// TwinCAT 3 PLC project MotionDriver
// ProgramVersion: 3.1.4026.20
// libraries:
//   Tc2_MC2, * (Beckhoff Automation GmbH)
//   Tc2_Standard, * (Beckhoff Automation GmbH)
//   Tc2_System, * (Beckhoff Automation GmbH)
// project tree:
//   GVLs/ gVar.TcGVL
//   / PlcTask.TcTTO
//   POUs/ AxisDriver.TcPOU
// real-time tasks:
//   TASK PlcTask: cycle T#1ms, priority 20, ADS port 350
// motion (NC):
//   TASK NC-Task 1 SAF: cycle T#500us, priority 1, ADS port 501
//   TASK NC-Task 1 SVB: cycle T#10ms, priority 8, ADS port 511
//   AXIS Axis 1 (id 1)
//     General: UnitName=Degree
//     Dynamic: AccelerationMaximum=500, DecelerationMaximum=500, Acceleration=300, Deceleration=300, Jerk=1300
//     Velo: Maximum=50
//     OtherSettings: AllowMotionCmdToSlave=true
//     encoder EncType=19
//       EncPara: MaxCount=#xffffffff
//     drive DrvType=16
//       DrvPara: MaxCount=#xffffffff, DriveControlDWord=#x00020000
//         Analog: VeloReferenz=50, TorqueSetpointScale=10, ScaleFactorActTorque=0.1
//         TimeComp: TaskDelayCycles=1
//     controller CtrType=1
//       CtrPara: PriorControlFactor=1
//         Observer: BandWidth=20
// I/O:
//   DEVICE IPC Master, AmsNetId 5.154.213.103.2.1
//     Drive 1 (CAP-NET-E) [CAP-NET-E]
// variable links:
//   NC-Task 1 SAF/Axes/Axis 1 <-> IPC Master/Drive 1 (CAP-NET-E)
//     Drive/Inputs/In/nState1 <-> TPDO 1 mapping parameter/Status Word
//     Drive/Inputs/In/nState2 <-> TPDO 1 mapping parameter/Status Word @bit 8
//     Drive/Inputs/In/nState4 @bit 1 <-> WcState/InputToggle
//     Drive/Inputs/In/nState4 <-> WcState/WcState
//     Drive/Inputs/In/nState5 <-> TPDO 1 mapping parameter/Modes of operation display
//     Drive/Outputs/Out/nCtrl1 <-> RPDO 1 mapping parameter/Control Word
//     Drive/Outputs/Out/nCtrl2 <-> RPDO 1 mapping parameter/Control Word @bit 8
//     Drive/Outputs/Out/nCtrl5 <-> RPDO 1 mapping parameter/Modes of operation
//     Drive/Outputs/Out/nDataOut1 <-> RPDO 1 mapping parameter/Target position
//     Drive/Outputs/Out/nDataOut2 <-> RPDO 1 mapping parameter/Target velocity
//     Enc/Inputs/In/nDataIn1 <-> TPDO 1 mapping parameter/Position actual value
//     Enc/Inputs/In/nDataIn7 <-> TPDO 1 mapping parameter/Velocity actual value
//     Enc/Inputs/In/nState4 @bit 1 <-> WcState/InputToggle
//     Enc/Inputs/In/nState4 <-> WcState/WcState
//   MotionDriver/MotionDriver Instance <-> NC-Task 1 SAF/Axes/Axis 1
//     PlcTask Inputs/gVar.gAxis1.NcToPlc <-> Outputs/ToPlc
//     PlcTask Outputs/gVar.gAxis1.PlcToNc <-> Inputs/FromPlc

CONFIGURATION MotionDriver
    RESOURCE PLC ON TwinCAT3
        TASK PlcTask(INTERVAL := T#1ms, PRIORITY := 20);
        PROGRAM AxisDriver WITH PlcTask : AxisDriver;
    END_RESOURCE
END_CONFIGURATION

// ---- GVLs/gVar.TcGVL
{attribute 'qualified_only'}
VAR_GLOBAL
	gAxis1 : AXIS_REF; // Axis reference linked to Motion Axis 1
	
    // Inputs from drive (monitoring)
    gStatusWord     : UINT;
    gPosAct         : DINT;
    gVelAct         : DINT;
    gModeDisp       : SINT;

    // Outputs to drive (use with care - see note below)
    gControlWord    : UINT;
    gTargetPos      : DINT;
    gTargetVel      : DINT;
    gModeCmd        : SINT;
END_VAR

// ---- POUs/AxisDriver.TcPOU
PROGRAM AxisDriver
VAR
    fbReset : MC_Reset;  // PLCopen reset
    fbPower : MC_Power;  // PLCopen enable power
    bEnable : BOOL := TRUE;
END_VAR

// Reset faults
fbReset(
    Axis := gVar.gAxis1,
    Execute := bEnable
);

// Enable drive
fbPower(
    Axis := gVar.gAxis1,
    Enable := bEnable,
    Enable_Positive := TRUE,
    Enable_Negative := TRUE
);

END_PROGRAM
